(* IEC 61131-3 sources: CoDeSysV3.5-Project_1-Sensor-monitoring-and-HMI-/examples, 4 files *)

(* ---- MEASURE_POINT (STRUCT).st ---- *)
//Структура опреативных параметров одной точки измерения температуры
TYPE MEASURE_POINT :
STRUCT
	//Название точки измерения
	wsPointName: WSTRING(20);
	//Текущее значение температуры
	rValue: REAL;
	//Код ошибки аналогового входа
	eStatus: Mx210Assistant.ANALOG_SENSOR_ERRORS;
	//Текстовое описание ошибки
	wsString: WSTRING;
	//Признак выхода значения за допустимые границы
	xOutOfLimits: BOOL;
	//Сигнал ошибки
	xAlarm: BOOL;
	//Экземпляр таймера, используемый для задержки генерации ошибки
	//Позволяет отфильтровать кртковременный выход значения за допустимую границу
	fbAlarmDelay: TON;
	//Экземпляр блока детектирования изменения кода ошибки
	fdStatusChange: StatusChange;
END_STRUCT
END_TYPE

(* ---- MEASURE_POINT_LIM (STRUCT).st ---- *)
TYPE MEASURE_POINT_LIM :
STRUCT
	//Нижняя предел температур
	rLowAlarmValur: REAL := 10.0;
	//Верхний прдел температур
	rHightAlarmValue: REAL := 30.0;
	//Экземпляр счётчика ошибок
	fbAlarmCounter: CTU;
END_STRUCT
END_TYPE

(* ---- StatusChange (FB).st ---- *)
FUNCTION_BLOCK StatusChange
VAR_INPUT
	eStatus: Mx210Assistant.ANALOG_SENSOR_ERRORS;
END_VAR
VAR_OUTPUT
	Q: BOOL;
END_VAR
VAR
	ePrevStatus:	Mx210Assistant.ANALOG_SENSOR_ERRORS;
END_VAR

//Область кода
IF eStatus <> ePrevStatus THEN
	Q := TRUE;
	ePrevStatus := eStatus;
ELSE
	Q := FALSE;
END_IF

(* ---- PLC_PRG (PRG).st ---- *)
PROGRAM PLC_PRG
VAR
	astMeasurePoints: ARRAY [1..c_iMeasureCount] OF MEASURE_POINT;
	i: INT;
	xInit: BOOL := FALSE;
	iCurrentFrameIndex: INT := 1;
	xEnableArchive: BOOL := TRUE;
END_VAR
VAR RETAIN
	astMeasurePointsLimit: ARRAY [1..c_iMeasureCount] OF MEASURE_POINT_LIM;
END_VAR
VAR CONSTANT
	c_iMeasureCount: INT := 8;
	c_iAlarmDelay: TIME := T#5S;
END_VAR

//Область кода

//Инициализация наименования точек измерения температуры
IF NOT(xInit) THEN
   astMeasurePoints[1].wsPointName := "Точка измерения 1";
   astMeasurePoints[2].wsPointName := "Точка измерения 2";
   astMeasurePoints[3].wsPointName := "Точка измерения 3";
   astMeasurePoints[4].wsPointName := "Точка измерения 4";
   astMeasurePoints[5].wsPointName := "Точка измерения 5";
   astMeasurePoints[6].wsPointName := "Точка измерения 6";
   astMeasurePoints[7].wsPointName := "Точка измерения 7";
   astMeasurePoints[8].wsPointName := "Точка измерения 8";
   xInit := TRUE;
END_IF

//Цикл обработки значений массива температур
FOR i := 1 TO c_iMeasureCount DO
	astMeasurePoints[i].xOutOfLimits := IsValueOutOfLimit(astMeasurePoints[i].rValue, astMeasurePointsLimit[i].rLowAlarmValur, astMeasurePointsLimit[i].rHightAlarmValue);
	astMeasurePoints[i].fbAlarmDelay
	(
		IN := astMeasurePoints[i].xOutOfLimits OR astMeasurePoints[i].eStatus <> Mx210Assistant.ANALOG_SENSOR_ERRORS.NO_ERROR,
		PT := c_iAlarmDelay,
		Q => astMeasurePoints[i].xAlarm
	);

	 astMeasurePointsLimit[i].fbAlarmCounter(CU := astMeasurePoints[i].xAlarm);

	 astMeasurePoints[i].fdStatusChange(eStatus := astMeasurePoints[i].eStatus);
	 IF astMeasurePoints[i].fdStatusChange.Q THEN
		 astMeasurePoints[i].wsString := Mx210Assistant.ANALOG_SENSOR_ERROR_TO_WSTRING(astMeasurePoints[i].eStatus);
	 END_IF

END_FOR
